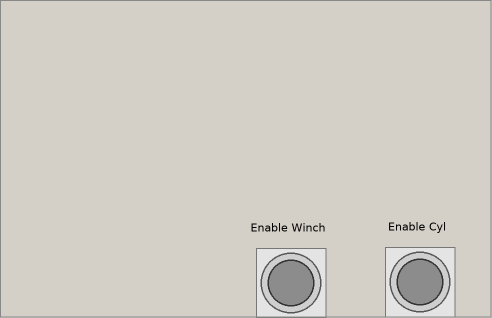
VISUALIZATION Visualization  // 492x318
    PushSwitch (256,248 70x70), variable: G_Hmi.bWinchEnable, behaviour: TOGGLE, style: Switch-PushSwitch-Gray
    Label (213,213 150x30), "Enable Winch"
    Label (342,212 150x30), "Enable Cyl"
    PushSwitch (385,247 70x70), variable: G_Hmi.bCylEnable, behaviour: TOGGLE, style: Switch-PushSwitch-Gray
END_VISUALIZATION

(* stored: Version 1.1.0.1, ProductVersion 3.1.4024.11
   Visu Visualization: Id {c8398d6f-4ceb-4850-a46d-48fbc6c4726c} *)
